// TIA Portal V19 export
DATA_BLOCK "DataFromSafety"   // DB127
// stored: Access Published, InstanceOfName Safety.typeDataFromSafety, InstanceOfType UDT, Namespace Safety
"Safety.typeDataFromSafety"
   // VAR
   //    safetyReleasedAllSafetyZones { ExternalWritable := 'False'} : Bool;
   //    ackRequiredAnySafetyZone { ExternalWritable := 'False'} : Bool;
   //    ackOP_changeRequired { ExternalWritable := 'False'} : Bool;
   //    devicesSummary { ExternalWritable := 'False'} : "Safety.typeDevicesStatusSummary";
   //    eStopButton0pressed { ExternalWritable := 'False'} : Bool;
   //    eStopButton1pressed { ExternalWritable := 'False'} : Bool;
   //    fDoor1Open { ExternalWritable := 'False'} : Bool;
   //    AOPD1interrupted { ExternalWritable := 'False'} : Bool;
   //    eStopZone1 { ExternalWritable := 'False'} : "Safety.typeEstopFunction";
   //    fDoorZone1 { ExternalWritable := 'False'} : "Safety.typeFDoorFunction";
   //    lightCurtainZone1 { ExternalWritable := 'False'} : "Safety.typeAOPD_Function";
   //    statusZone1 { ExternalWritable := 'False'} : "Safety.typeSafetyZoneStatus";
   //    activeSTO_Zone1 { ExternalWritable := 'False'} : Bool;
   //    drive1 { ExternalWritable := 'False'} : "Safety.typeSafetyDrive";
   //    drive2 { ExternalWritable := 'False'} : "Safety.typeSafetyDrive";
   // END_VAR
BEGIN
   // statusZone1.safetyReleased : Zone 1 not released / Safety Zone 3 nicht freigegeben
   // statusZone1.ackReq : Zone 1 : Acknowledge required / Safety Zone 3 : Acknowledge oder Clear erforderlich
END_DATA_BLOCK
